// TIA Portal V20 export
TYPE "UDT_EmisionDeDispositivo"
   STRUCT
      Error : UDInt;
      Auxliar_01 : UInt;
      Auxliar_02 : UInt;
      Protocolo { S7_SetPoint := 'True'} : "UDT_ProtocoloEmiDispositivo";
   END_STRUCT;
END_TYPE
